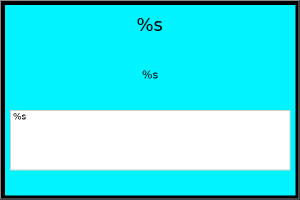
VISUALIZATION VISU_BUS_DIAG_MASTER  // 300x200
VAR_IN_OUT
	fbVisu: FB_VISU_BUS_DIAG;
END_VAR
    Rectangle (0,0 300x200), colour variable: fbVisu.dwColor
        p3450524324: fbVisu.dwColorFrame
    Textfield (10,10 280x30), "%s", text variable: fbVisu.strType
    Textfield (10,60 280x30), "%s", text variable: fbVisu.strName
    Textfield (10,110 280x60), "%s", text variable: fbVisu.strState
END_VISUALIZATION

(* stored: Version 1.1.0.1, ProductVersion 3.1.4024.4
   Visu VISU_BUS_DIAG_MASTER: Id {34bc1065-7949-40b3-91f9-c82d52d45452} *)
